TYPE
   stEL9410 :
   STRUCT
      Us_Undervoltage AT %I* : BIT;
      Up_Undervoltage AT %I* : BIT;
   END_STRUCT
END_TYPE

(* stored: Version 1.1.0.1, ProductVersion 3.1.4024.9
   DUT stEL9410: Id {cc93f896-e3c8-45b7-ba50-84ee95b8cf4a} *)
